TYPE HMI_STS_General :
STRUCT
	Version:STRING(23);								//Project version
END_STRUCT
END_TYPE

(* stored: Version 1.1.0.1
   DUT HMI_STS_General: Id {e72b8229-4b31-4714-9921-2a9712bfb4fa} *)
